// Mitsubishi GX Works2 project: pro14   PLC: FX3G

// global labels: Global1
VAR_GLOBAL
  start AT X007 : BOOL;
  analog_input1 AT D8280 : INT;
  numOfPack AT D1112 : REAL;
  analog_output AT D8282 : INT;
  job1 AT X001 : BOOL;
  is_pinuk AT M3 : BOOL;
  is_ragil AT M4 : BOOL;
  lemon_inv AT D3333 : REAL;
  petel_inv AT D4444 : REAL;
  meshamer_inv AT D5555 : REAL;
  gumi_inv AT D6666 : REAL;
END_VAR
VAR_GLOBAL CONSTANT
  pinuk_lemon : REAL := 665;
  pinuk_petel : REAL := 385;
  pinuk_meshamer : REAL := 210;
  pink_gumi : REAL := 70;
  ragil_lemon : REAL := 455;
  ragil_petel : REAL := 280;
  ragil_meshamer : REAL := 105;
  ragil_gumi : REAL := 28;
END_VAR
VAR_GLOBAL
  pinuk_check AT M55 : BOOL;
  ragil_check AT M6 : BOOL;
END_VAR
VAR_GLOBAL CONSTANT
  normalization : REAL := 400;
  const1 : REAL := 5;
  const2 : REAL := 10;
  const3 : REAL := 6;
END_VAR
VAR_GLOBAL
  day_finish_pinuk AT M7 : BOOL;
  day_finish_ragil AT M8 : BOOL;
  no_initial_stock AT M9 : BOOL;
  not_day_finish AT M10 : BOOL;
  during_day AT Y007 : BOOL;
  emergency AT X005 : BOOL;
  fishing_making_pinuk AT M11 : BOOL;
  fishing_making_ragil AT M12 : BOOL;
  timer_when_making AT TS1 : BOOL;
  lamp_making AT Y000 : BOOL;
  TC AT TC1 : BOOL;
END_VAR
VAR_GLOBAL CONSTANT
  timer_making : INT := 50;
  pinuk_petel_to_petel : REAL := 385;
  pinuk_meshamer_to_petel : REAL := 70;
END_VAR
VAR_GLOBAL
  reg_petel AT D2111 : REAL;
END_VAR
VAR_GLOBAL CONSTANT
  pinuk_lemon_to_lemon : REAL := 560;
  pinuk_meshamer_to_lemon : REAL := 140;
END_VAR
VAR_GLOBAL
  reg_lemon AT D3111 : REAL;
END_VAR
VAR_GLOBAL CONSTANT
  ragil_petel_to_petel : REAL := 280;
  ragil_lemon_to_petel : REAL := 35;
  ragil_meshamer_to_petel : REAL := 35;
  ragil_lemon_to_lemon : REAL := 420;
  ragil_meshamer_to_lemon : REAL := 70;
END_VAR
VAR_GLOBAL
  move_icecream AT X002 : BOOL;
  cooling_petel AT D4111 : REAL;
  cooling_lemon AT D5111 : REAL;
  start_cooling AT M13 : BOOL;
  temp_sensor AT X003 : BOOL;
  TC_2 AT TC2 : BOOL;
END_VAR
VAR_GLOBAL CONSTANT
  timer_cooling : INT := 80;
END_VAR
VAR_GLOBAL
  timer_when_cooling AT TS2 : BOOL;
  lamp_cooling AT Y002 : BOOL;
END_VAR
VAR_GLOBAL CONSTANT
  pinuk_lemon_to_petel : REAL := 105;
END_VAR
VAR_GLOBAL
  lemon_input AT D3344 : REAL;
  petel : BOOL;
  petel_input AT D3355 : REAL;
  meshamer_input AT D3366 : REAL;
  gumi_input AT D3377 : REAL;
  is_ragil_help AT M41 : BOOL;
  is_pinuk_help AT M31 : BOOL;
  pinuk_check_help AT M51 : BOOL;
  ragil_check_help AT M61 : BOOL;
  reset_lamp AT M100 : BOOL;
  packing AT Y004 : BOOL;
  mixing_reg AT D6111 : REAL;
  start_making_pinuk AT M11 : BOOL;
END_VAR
VAR_GLOBAL CONSTANT
  add_gumi_pinuk : REAL := 70;
END_VAR
VAR_GLOBAL
  start_making_ragil AT M12 : BOOL;
END_VAR
VAR_GLOBAL CONSTANT
  add_gumi_ragil : REAL := 28;
END_VAR
VAR_GLOBAL
  start_mixing AT M14 : BOOL;
  mixing_ragil AT TC4 : BOOL;
END_VAR
VAR_GLOBAL CONSTANT
  time_mixing_ragil : INT := 30;
END_VAR
VAR_GLOBAL
  mixing_pinuk AT TC3 : BOOL;
END_VAR
VAR_GLOBAL CONSTANT
  time_mixing_pinuk : INT := 50;
END_VAR
VAR_GLOBAL
  finish_mixing_pinuk AT TS3 : BOOL;
  finish_mixing_ragil AT TS4 : BOOL;
  M_100 AT M100 : BOOL;
  y5_blink AT TS5 : BOOL;
  y5_timer AT TC5 : BOOL;
END_VAR
VAR_GLOBAL CONSTANT
  y5_time : INT := 5;
END_VAR
VAR_GLOBAL
  y_5 AT Y005 : BOOL;
  y6_blink AT TS6 : BOOL;
  y6_timer AT TC6 : BOOL;
END_VAR
VAR_GLOBAL CONSTANT
  y6_time : INT := 5;
END_VAR
VAR_GLOBAL
  y_6 AT Y006 : BOOL;
  start_packing AT X004 : BOOL;
  one_gumigam AT X000 : BOOL;
  cone_counter AT CC1 : BOOL;
END_VAR
VAR_GLOBAL CONSTANT
  cones_in_package : WORD := 7;
END_VAR
VAR_GLOBAL
  finish_package AT CS1 : BOOL;
END_VAR
VAR_GLOBAL CONSTANT
  one_package : REAL := 1;
  add_0 : REAL;
END_VAR
VAR_GLOBAL
  M_101 AT M101 : BOOL;
  reset AT Y004 : BOOL;
  start_making_pinuk_help AT M16 : BOOL;
  reset_la AT M100 : BOOL;
  start_making_ragil_help AT M17 : BOOL;
  Output AT D8282 : INT;
END_VAR
VAR_GLOBAL CONSTANT
  zero : REAL;
  zero_word : INT;
END_VAR
VAR_GLOBAL
  next_day AT M125 : BOOL;
END_VAR
VAR_GLOBAL CONSTANT
  numOfPack_norm : REAL := 40;
END_VAR

// task Task_01 (event TRUE, interval 0, priority 31): POU_01

PROGRAM POU_01
(* structured ladder/FBD written out as ST: instructions are called as NAME(EN, inputs, outputs); _pN, _eN, _tN stand for wires *)
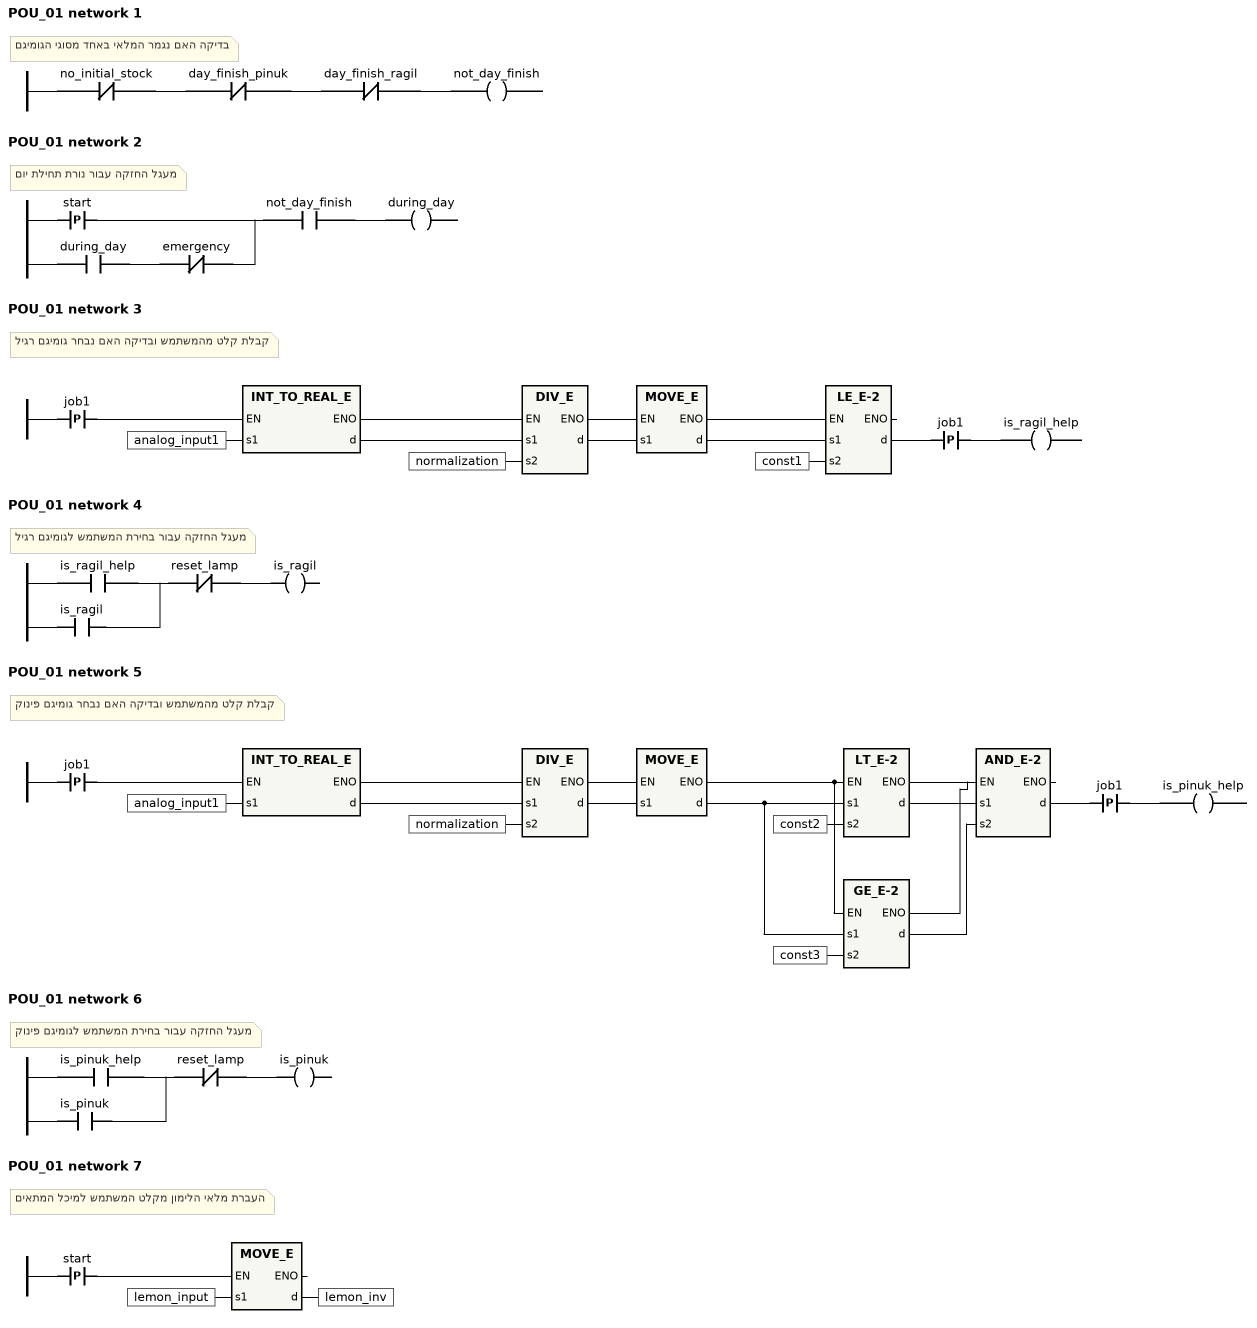
(* network 1 *)
(* בדיקה האם נגמר המלאי באחד מסוגי הגומיגם *)
not_day_finish := NOT no_initial_stock AND NOT day_finish_pinuk AND NOT day_finish_ragil;
(* network 2 *)
(* מעגל החזקה עבור נורת תחילת יום *)
during_day := (LDP(TRUE, start) OR (during_day AND NOT emergency)) AND not_day_finish;
(* network 3 *)
(* קבלת קלט מהמשתמש ובדיקה האם נבחר גומיגם רגיל *)
_e2 := INT_TO_REAL_E(LDP(TRUE, job1), analog_input1, _t1);
_e4 := DIV_E(_e2, _t1, normalization, _t3);
_e6 := MOVE_E(_e4, _t3, _t5);
LE_E(_e6, _t5, const1, _t7);
is_ragil_help := _t7 AND LDP(TRUE, job1);
(* network 4 *)
(* מעגל החזקה עבור בחירת המשתמש לגומיגם רגיל *)
is_ragil := (is_ragil_help OR is_ragil) AND NOT reset_lamp;
(* network 5 *)
(* קבלת קלט מהמשתמש ובדיקה האם נבחר גומיגם פינוק *)
_e2 := INT_TO_REAL_E(LDP(TRUE, job1), analog_input1, _t1);
_e4 := DIV_E(_e2, _t1, normalization, _t3);
_e6 := MOVE_E(_e4, _t3, _t5);
_e8 := LT_E(_e6, _t5, const2, _t7);
_e10 := GE_E(_e6, _t5, const3, _t9);
AND_E(_e8 OR _e10, _t7, _t9, _t11);
is_pinuk_help := _t11 AND LDP(TRUE, job1);
(* network 6 *)
(* מעגל החזקה עבור בחירת המשתמש לגומיגם פינוק *)
is_pinuk := (is_pinuk_help OR is_pinuk) AND NOT reset_lamp;
(* network 7 *)
(* העברת מלאי הלימון מקלט המשתמש למיכל המתאים *)
MOVE_E(LDP(TRUE, start), lemon_input, lemon_inv);
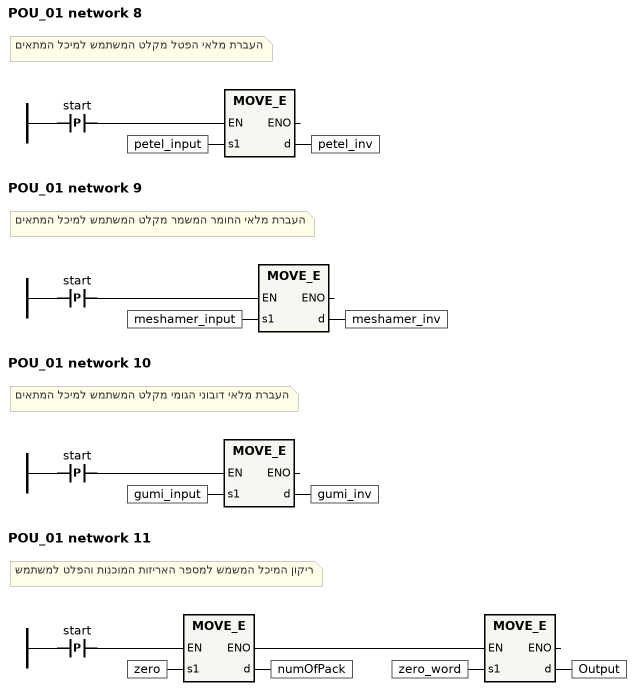
(* network 8 *)
(* העברת מלאי הפטל מקלט המשתמש למיכל המתאים *)
MOVE_E(LDP(TRUE, start), petel_input, petel_inv);
(* network 9 *)
(* העברת מלאי החומר המשמר מקלט המשתמש למיכל המתאים *)
MOVE_E(LDP(TRUE, start), meshamer_input, meshamer_inv);
(* network 10 *)
(* העברת מלאי דובוני הגומי מקלט המשתמש למיכל המתאים *)
MOVE_E(LDP(TRUE, start), gumi_input, gumi_inv);
(* network 11 *)
(* ריקון המיכל המשמש למספר האריזות המוכנות והפלט למשתמש *)
_e1 := MOVE_E(LDP(TRUE, start), zero, numOfPack);
MOVE_E(_e1, zero_word, Output);
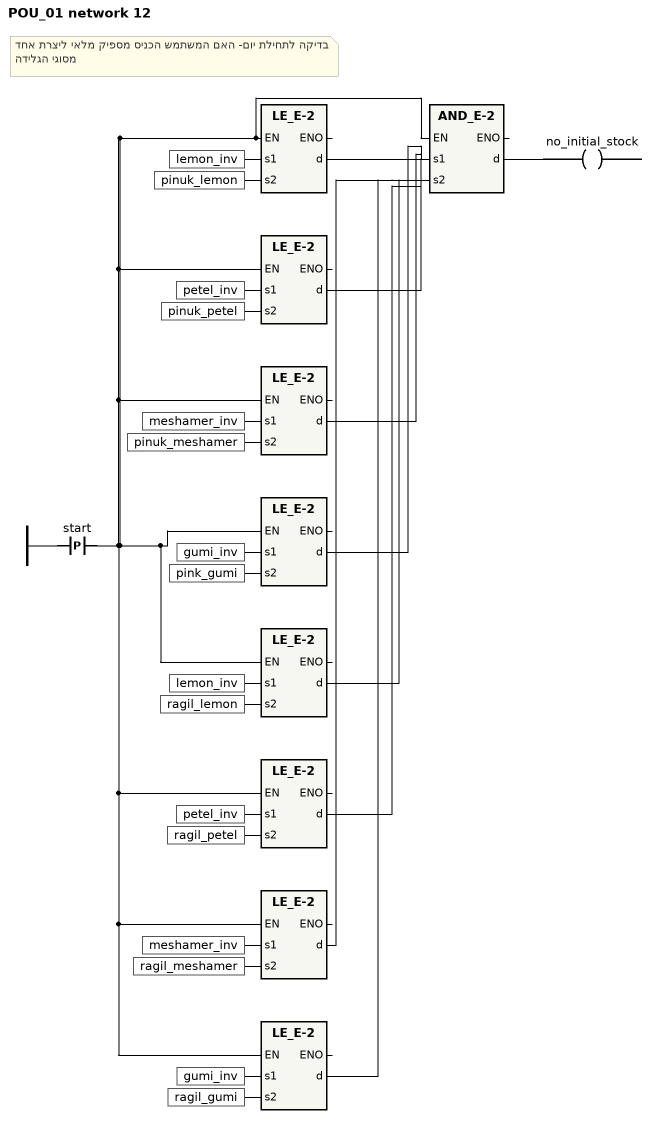
(* network 12 *)
(* בדיקה לתחילת יום- האם המשתמש הכניס מספיק מלאי ליצרת אחד מסוגי הגלידה *)
_p1 := LDP(TRUE, start);
LE_E(_p1, lemon_inv, pinuk_lemon, _t2);
LE_E(_p1, petel_inv, pinuk_petel, _t3);
LE_E(_p1, meshamer_inv, pinuk_meshamer, _t4);
LE_E(_p1, gumi_inv, pink_gumi, _t5);
LE_E(_p1, lemon_inv, ragil_lemon, _t6);
LE_E(_p1, petel_inv, ragil_petel, _t7);
LE_E(_p1, meshamer_inv, ragil_meshamer, _t8);
LE_E(_p1, gumi_inv, ragil_gumi, _t9);
AND_E(_p1, _t2 OR _t3 OR _t4 OR _t5, _t6 OR _t7 OR _t8 OR _t9, _t10);
no_initial_stock := _t10;
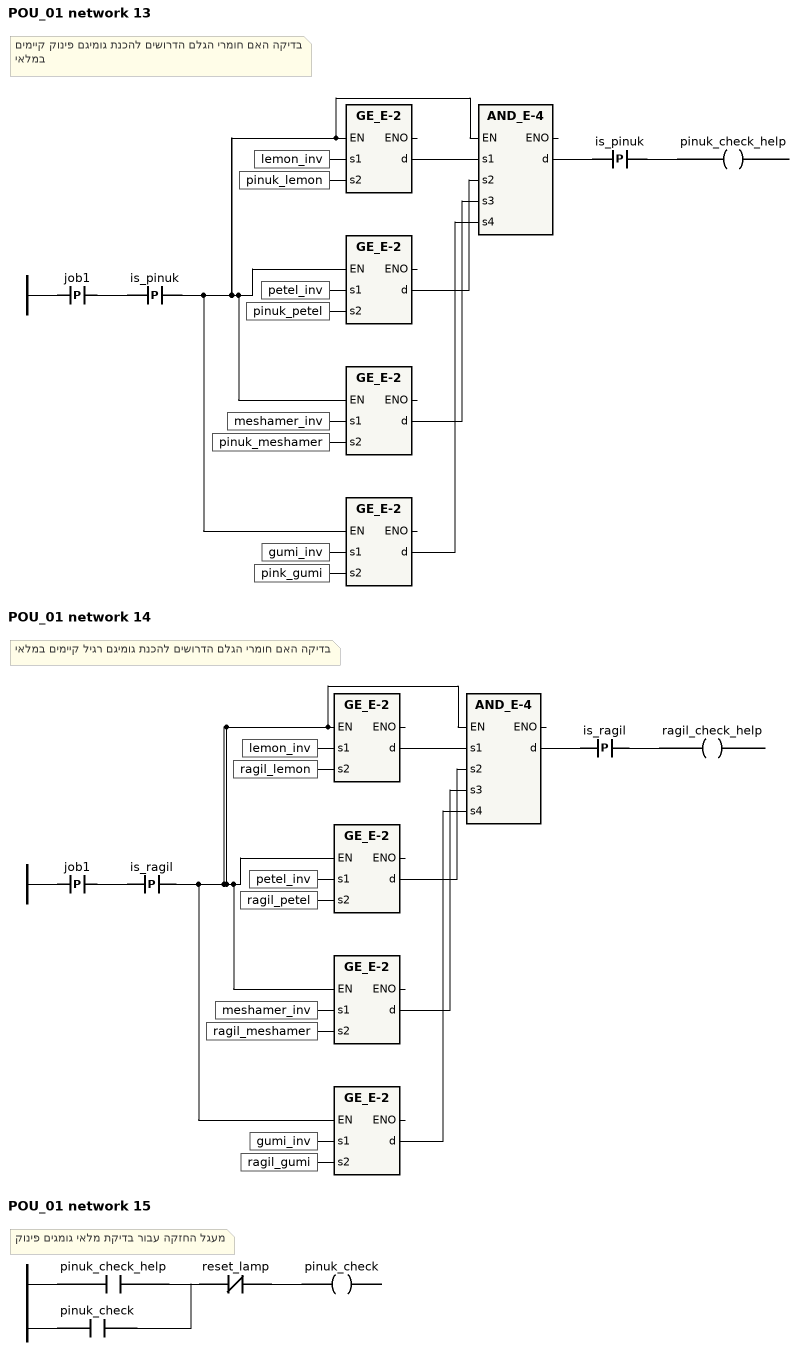
(* network 13 *)
(* בדיקה האם חומרי הגלם הדרושים להכנת גומיגם פינוק קיימים במלאי *)
_p1 := LDP(TRUE, job1) AND LDP(TRUE, is_pinuk);
GE_E(_p1, lemon_inv, pinuk_lemon, _t2);
GE_E(_p1, petel_inv, pinuk_petel, _t3);
GE_E(_p1, meshamer_inv, pinuk_meshamer, _t4);
GE_E(_p1, gumi_inv, pink_gumi, _t5);
AND_E(_p1, _t2, _t3, _t4, _t5, _t6);
pinuk_check_help := _t6 AND LDP(TRUE, is_pinuk);
(* network 14 *)
(* בדיקה האם חומרי הגלם הדרושים להכנת גומיגם רגיל קיימים במלאי *)
_p1 := LDP(TRUE, job1) AND LDP(TRUE, is_ragil);
GE_E(_p1, lemon_inv, ragil_lemon, _t2);
GE_E(_p1, petel_inv, ragil_petel, _t3);
GE_E(_p1, meshamer_inv, ragil_meshamer, _t4);
GE_E(_p1, gumi_inv, ragil_gumi, _t5);
AND_E(_p1, _t2, _t3, _t4, _t5, _t6);
ragil_check_help := _t6 AND LDP(TRUE, is_ragil);
(* network 15 *)
(* מעגל החזקה עבור בדיקת מלאי גומגים פינוק *)
pinuk_check := (pinuk_check_help OR pinuk_check) AND NOT reset_lamp;
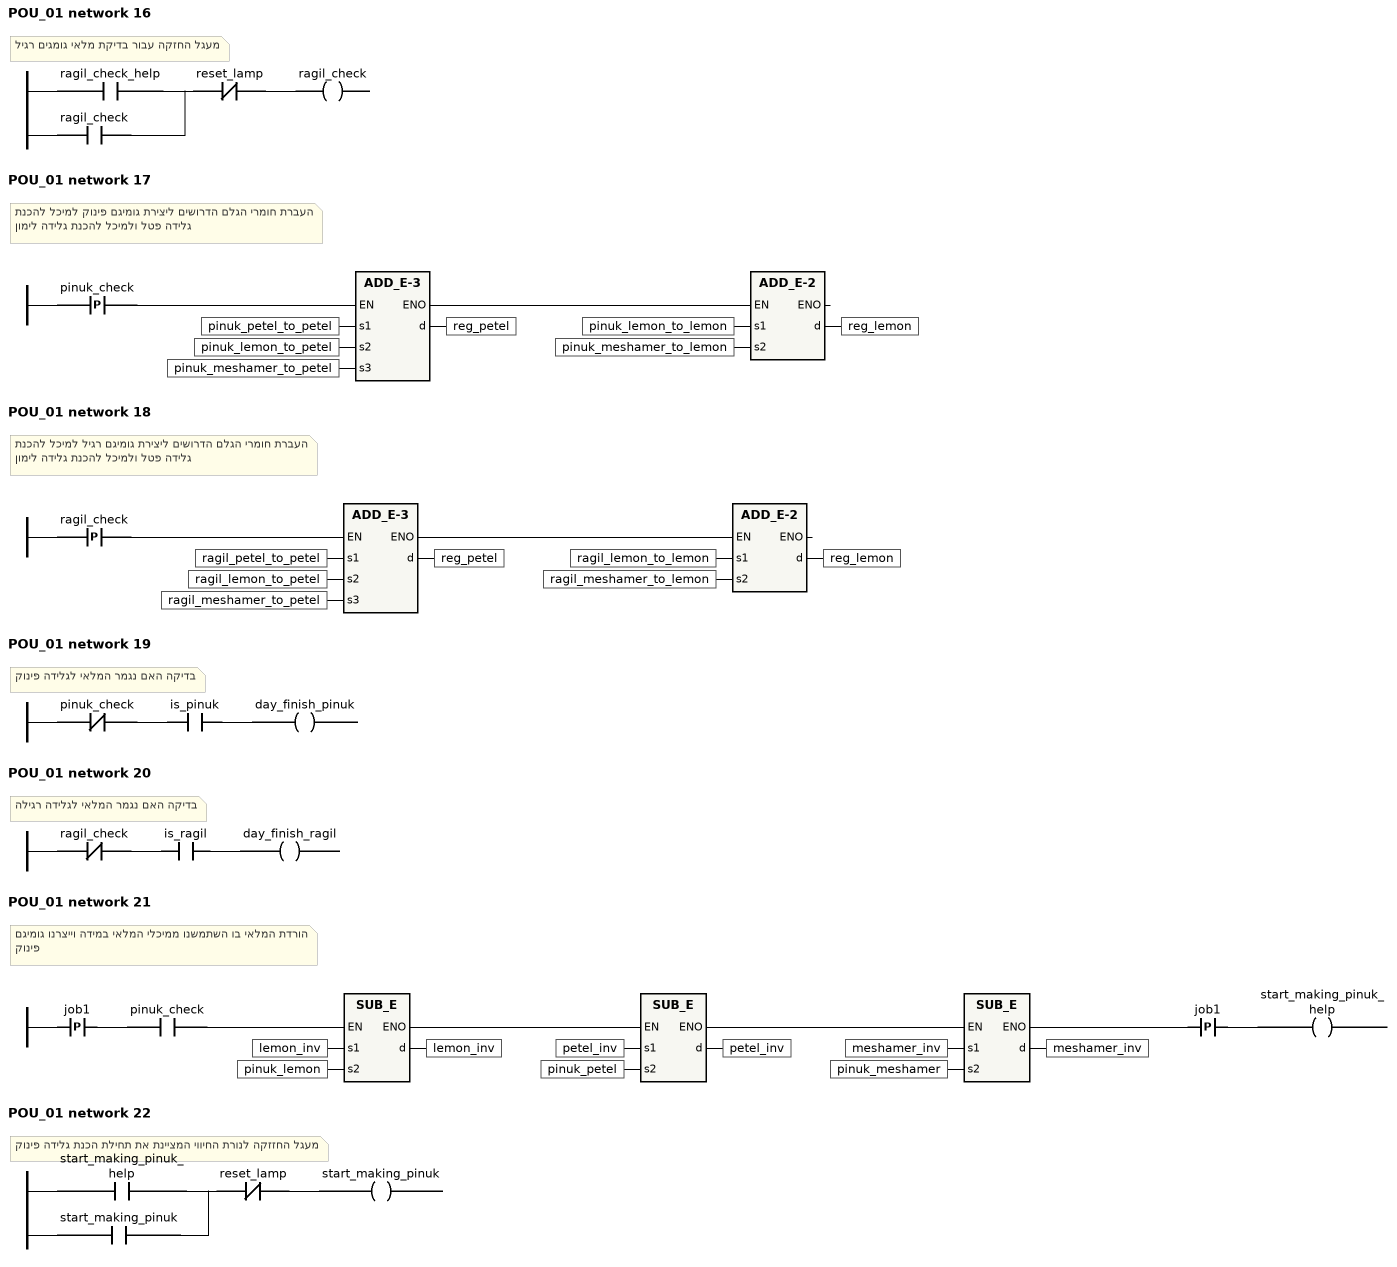
(* network 16 *)
(* מעגל החזקה עבור בדיקת מלאי גומגים רגיל *)
ragil_check := (ragil_check_help OR ragil_check) AND NOT reset_lamp;
(* network 17 *)
(* העברת חומרי הגלם הדרושים ליצירת גומיגם פינוק למיכל להכנת גלידה פטל ולמיכל להכנת גלידה לימון *)
_e1 := ADD_E(LDP(TRUE, pinuk_check), pinuk_petel_to_petel, pinuk_lemon_to_petel, pinuk_meshamer_to_petel, reg_petel);
ADD_E(_e1, pinuk_lemon_to_lemon, pinuk_meshamer_to_lemon, reg_lemon);
(* network 18 *)
(* העברת חומרי הגלם הדרושים ליצירת גומיגם רגיל למיכל להכנת גלידה פטל ולמיכל להכנת גלידה לימון *)
_e1 := ADD_E(LDP(TRUE, ragil_check), ragil_petel_to_petel, ragil_lemon_to_petel, ragil_meshamer_to_petel, reg_petel);
ADD_E(_e1, ragil_lemon_to_lemon, ragil_meshamer_to_lemon, reg_lemon);
(* network 19 *)
(* בדיקה האם נגמר המלאי לגלידה פינוק *)
day_finish_pinuk := NOT pinuk_check AND is_pinuk;
(* network 20 *)
(* בדיקה האם נגמר המלאי לגלידה רגילה *)
day_finish_ragil := NOT ragil_check AND is_ragil;
(* network 21 *)
(* הורדת המלאי בו השתמשנו ממיכלי המלאי במידה וייצרנו גומיגם פינוק *)
_e1 := SUB_E(LDP(TRUE, job1) AND pinuk_check, lemon_inv, pinuk_lemon, lemon_inv);
_e2 := SUB_E(_e1, petel_inv, pinuk_petel, petel_inv);
_e3 := SUB_E(_e2, meshamer_inv, pinuk_meshamer, meshamer_inv);
start_making_pinuk_help := _e3 AND LDP(TRUE, job1);
(* network 22 *)
(* מעגל החזזקה לנורת החיווי המציינת את תחילת הכנת גלידה פינוק *)
start_making_pinuk := (start_making_pinuk_help OR start_making_pinuk) AND NOT reset_lamp;
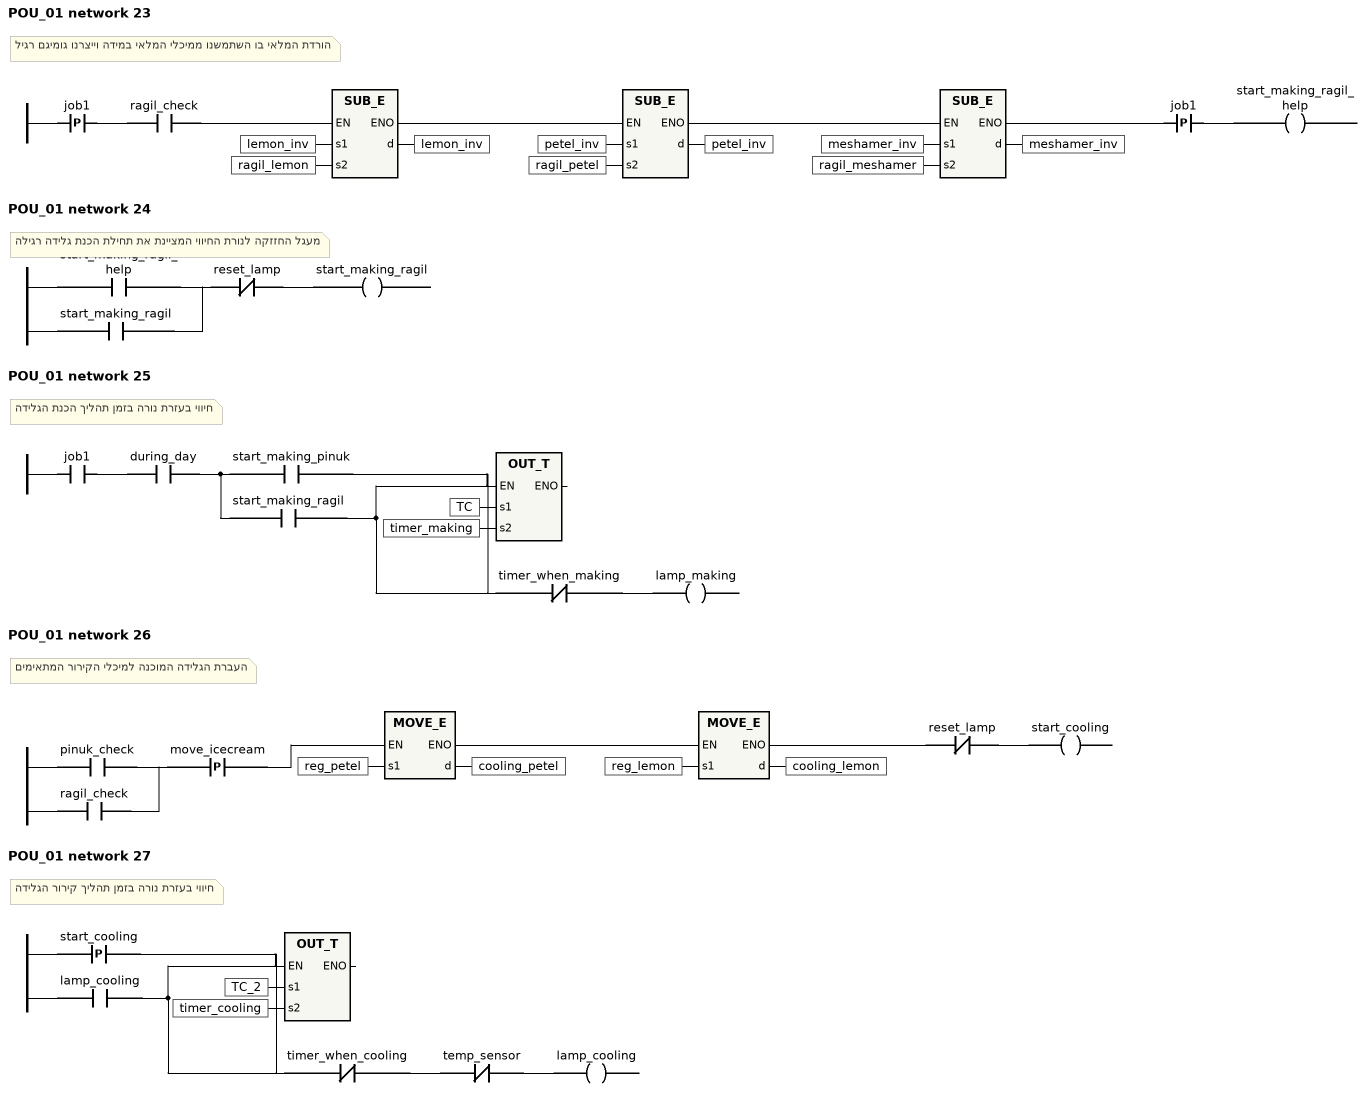
(* network 23 *)
(* הורדת המלאי בו השתמשנו ממיכלי המלאי במידה וייצרנו גומיגם רגיל *)
_e1 := SUB_E(LDP(TRUE, job1) AND ragil_check, lemon_inv, ragil_lemon, lemon_inv);
_e2 := SUB_E(_e1, petel_inv, ragil_petel, petel_inv);
_e3 := SUB_E(_e2, meshamer_inv, ragil_meshamer, meshamer_inv);
start_making_ragil_help := _e3 AND LDP(TRUE, job1);
(* network 24 *)
(* מעגל החזזקה לנורת החיווי המציינת את תחילת הכנת גלידה רגילה *)
start_making_ragil := (start_making_ragil_help OR start_making_ragil) AND NOT reset_lamp;
(* network 25 *)
(* חיווי בעזרת נורה בזמן תהליך הכנת הגלידה *)
_p1 := job1 AND during_day;
_p2 := (_p1 AND start_making_pinuk) OR (_p1 AND start_making_ragil);
lamp_making := _p2 AND NOT timer_when_making;
OUT_T(_p2, TC, timer_making);
(* network 26 *)
(* העברת הגלידה המוכנה למיכלי הקירור המתאימים *)
_e1 := MOVE_E((pinuk_check OR ragil_check) AND LDP(TRUE, move_icecream), reg_petel, cooling_petel);
_e2 := MOVE_E(_e1, reg_lemon, cooling_lemon);
start_cooling := _e2 AND NOT reset_lamp;
(* network 27 *)
(* חיווי בעזרת נורה בזמן תהליך קירור הגלידה *)
_p1 := LDP(TRUE, start_cooling) OR lamp_cooling;
lamp_cooling := _p1 AND NOT timer_when_cooling AND NOT temp_sensor;
OUT_T(_p1, TC_2, timer_cooling);
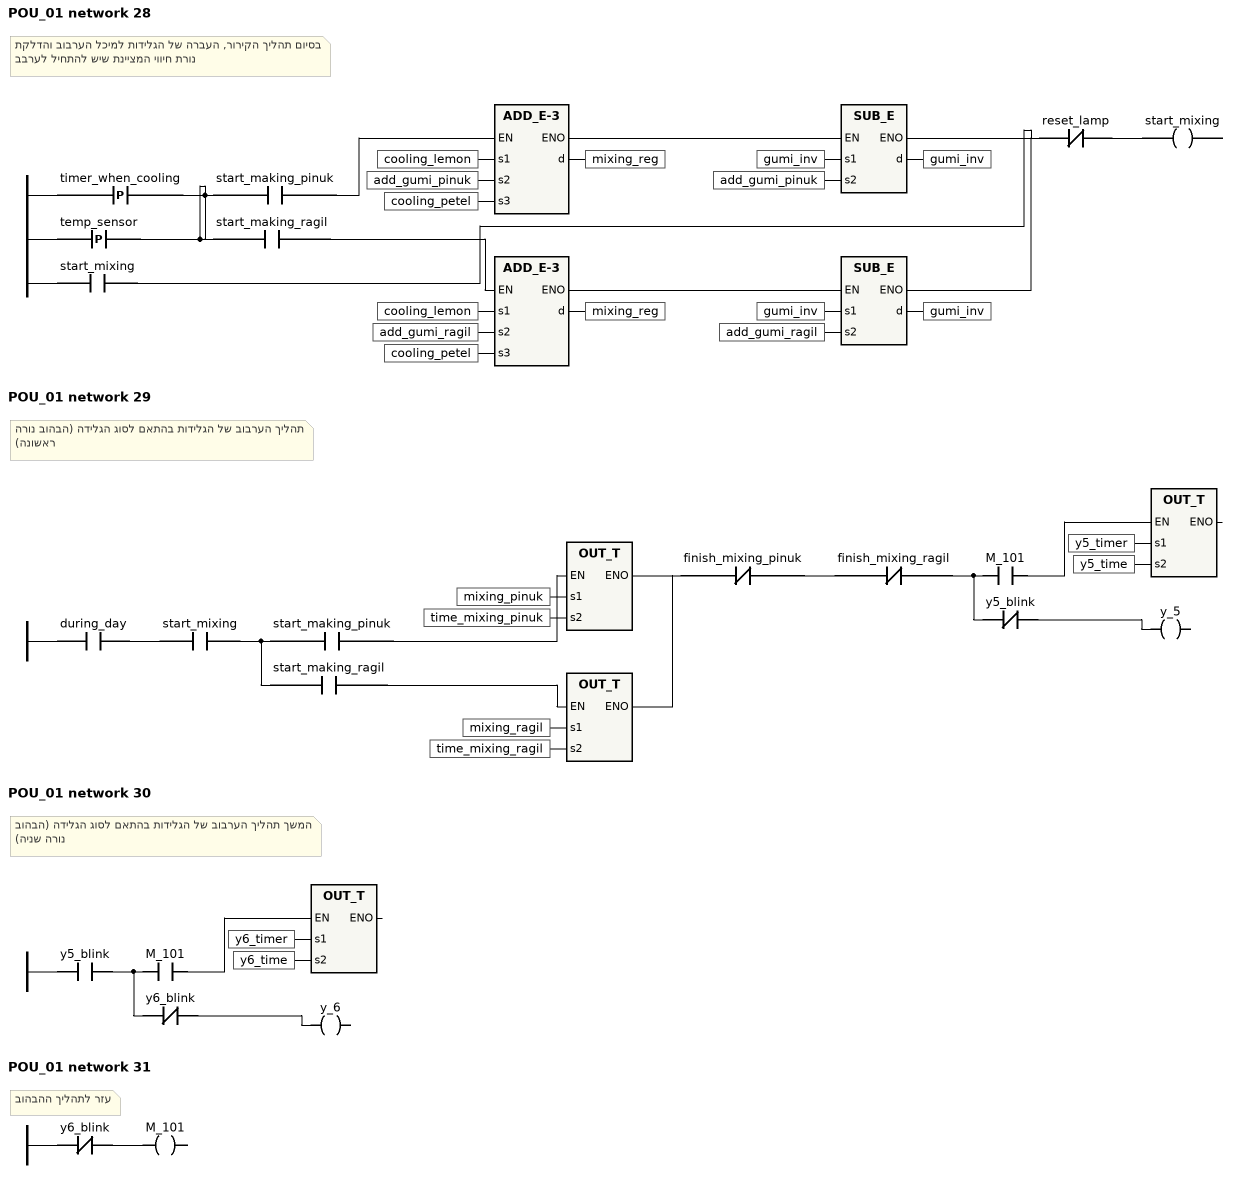
(* network 28 *)
(* בסיום תהליך הקירור, העברה של הגלידות למיכל הערבוב והדלקת נורת חיווי המציינת שיש להתחיל לערבב *)
_p1 := LDP(TRUE, timer_when_cooling) OR LDP(TRUE, temp_sensor);
_e2 := ADD_E(_p1 AND start_making_pinuk, cooling_lemon, add_gumi_pinuk, cooling_petel, mixing_reg);
_e3 := SUB_E(_e2, gumi_inv, add_gumi_pinuk, gumi_inv);
_e4 := ADD_E(_p1 AND start_making_ragil, cooling_lemon, add_gumi_ragil, cooling_petel, mixing_reg);
_e5 := SUB_E(_e4, gumi_inv, add_gumi_ragil, gumi_inv);
start_mixing := (_e3 OR _e5 OR start_mixing) AND NOT reset_lamp;
(* network 29 *)
(* תהליך הערבוב של הגלידות בהתאם לסוג הגלידה (הבהוב נורה ראשונה) *)
_p1 := during_day AND start_mixing;
_e2 := OUT_T(_p1 AND start_making_pinuk, mixing_pinuk, time_mixing_pinuk);
_e3 := OUT_T(_p1 AND start_making_ragil, mixing_ragil, time_mixing_ragil);
_p4 := ((_e2 OR _e3) AND NOT finish_mixing_pinuk) AND NOT finish_mixing_ragil;
OUT_T(_p4 AND M_101, y5_timer, y5_time);
y_5 := _p4 AND NOT y5_blink;
(* network 30 *)
(* המשך תהליך הערבוב של הגלידות בהתאם לסוג הגלידה (הבהוב נורה שניה) *)
OUT_T(y5_blink AND M_101, y6_timer, y6_time);
y_6 := y5_blink AND NOT y6_blink;
(* network 31 *)
(* עזר לתהליך ההבהוב *)
M_101 := NOT y6_blink;
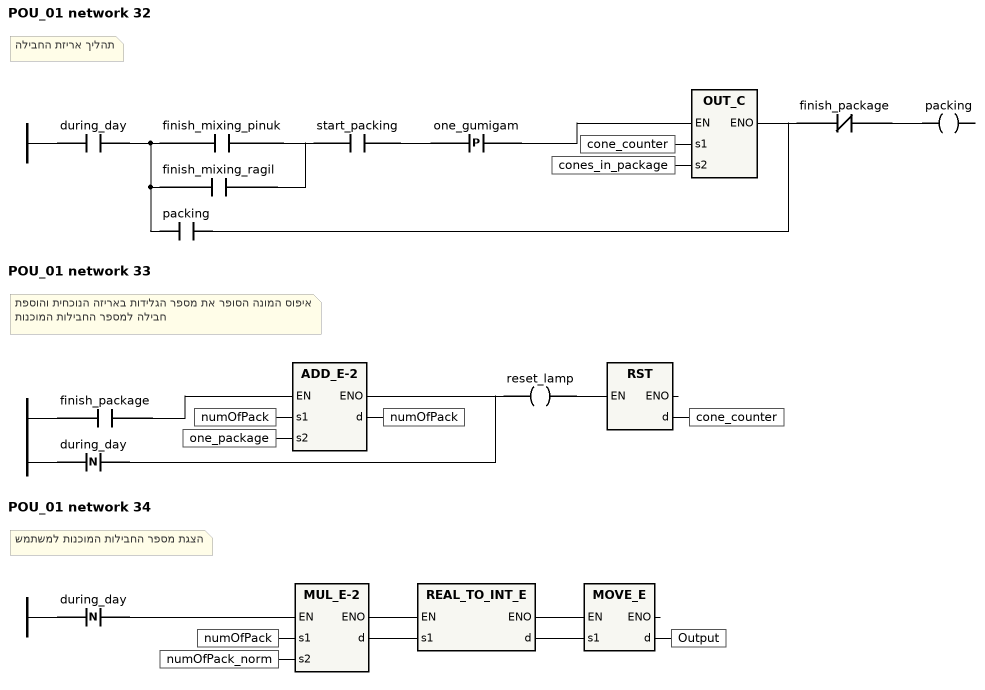
(* network 32 *)
(* תהליך אריזת החבילה *)
_e1 := OUT_C((((during_day AND finish_mixing_pinuk) OR (during_day AND finish_mixing_ragil)) AND start_packing) AND LDP(TRUE, one_gumigam), cone_counter, cones_in_package);
packing := (_e1 OR (during_day AND packing)) AND NOT finish_package;
(* network 33 *)
(* איפוס המונה הסופר את מספר הגלידות באריזה הנוכחית והוספת חבילה למספר החבילות המוכנות *)
_e1 := ADD_E(finish_package, numOfPack, one_package, numOfPack);
_p2 := _e1 OR LDF(TRUE, during_day);
reset_lamp := _p2;
RST(_p2, cone_counter);
(* network 34 *)
(* הצגת מספר החבילות המוכנות למשתמש *)
_e2 := MUL_E(LDF(TRUE, during_day), numOfPack, numOfPack_norm, _t1);
_e4 := REAL_TO_INT_E(_e2, _t1, _t3);
MOVE_E(_e4, _t3, Output);
END_PROGRAM
